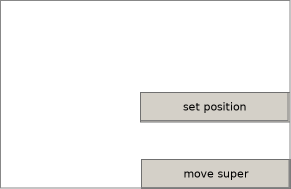
VISUALIZATION superimposed  // 291x189
    Button (140,92 150x30), "set position", colour toggle: superimpose.shouldSetPosition
        tap superimpose.shouldSetPosition
    Button (141,159 150x30), "move super", colour toggle: superimpose.shouldMoveVelocity
        tap superimpose.shouldMoveVelocity
END_VISUALIZATION

(* stored: Version 1.1.0.1, ProductVersion 3.1.4024.4
   Visu superimposed: Id {0f328fac-98d0-4e25-b6c4-c5cdcba1344e} *)
